# EPICS alarm handler configuration: mps_database/bare/alarms/areas/mpln_spd_mp02.alhConfig
GROUP NULL MPLN:SPD:MP02:1
$ALIAS MPS Link Node 93
$GUIDANCE
LTUH MPS
   Group Name: MPLN:SPD:MP02:1
   Summary PV:  MPLN:SPD:MP02:1:STATSUMY
$END
CHANNEL  MPLN:SPD:MP02:1    MPLN:SPD:MP02:1:MPS_EN_RBV		-----
CHANNEL  MPLN:SPD:MP02:1    MPLN:SPD:MP02:1:LC1_MODE_RBV		-----
